FUNCTION ifExprFunc1: DINT
VAR_INPUT
    farg_fac_a: DINT;
END_VAR

IF ((farg_fac_a) = (0)) THEN
    ifExprFunc1 := 1;
ELSE
    ifExprFunc1 := (func_fac((farg_fac_a) - (1))) * (farg_fac_a);
END_IF;

END_FUNCTION

(* stored: ProductVersion 3.1.0.18, Version 1.1.0.1 *)
